PROGRAM MAIN
VAR_OUTPUT //globally readable, but only modifiable by MAIN
	outputBuffer : ARRAY[Surface.LEFT..Surface.RIGHT] OF Bundle;
	outputBufferPass, outputBufferFail : Bundle;
	numOutputBundles : USINT := 0;
	
	bundleIn : Bundle;
	bundleOut : Bundle;
	
	start : BOOL;
	
	ready : BOOL;
	busy : BOOL;
	done : BOOL;
	error : BOOL;
	backlog : BOOL;
	
	stop : BOOL;
	execute : BOOL;
	hold : BOOL;
	reset : BOOL;
	
	localTime : TIMESTRUCT;
	
	pmlModeString : STRING;
	pmlStateString : STRING;
END_VAR
VAR
	clearPassBuffer, clearFailBuffer AT %I* : BOOL;
	receiverStruct : AdsData;
	
	//ETA is not strictly required, area will process bundle even if it is not in ETA arrays
	expectedBundles : ARRAY[0..GVL.maxQueue] OF STRING; //bundles expected to arrive
	expectedArrivals : ARRAY[0..GVL.maxQueue] OF TIMESTRUCT; //bundles expected to arrive
	numEtaBundles : INT;
	
	//parallel arrays - bundle, bypass
	numBundles : INT;
	bundlesQueue : ARRAY[0..GVL.maxQueue] OF Bundle;
	bundlesBypass : ARRAY[0..GVL.maxQueue] OF BOOL;
END_VAR
VAR
	//spacerRecollector : PackagerFreeAsync;
	//paperSection : PaperEx;
	//cardboardCornerGuardSection : CardboardCornerGuardEx;
	//chipboardSection : ChipboardEx;
	woodBunkSection : WoodBunkEx;
	//outputSection : AreaOutputEx;	
END_VAR
VAR
	fbLocalSystemTime : FB_LocalSystemTime;
	dbLogger : SqlDatabaseAccessor;
	conveyorController : ConveyorControlUnit;
	
	pmlState : E_PMLState;
	pmlCommand : E_PMLCommand;
	pmlStateMachine : PML_StateMachine;
	
	pmlModeRequest : E_PMLCustomUnitMode := ePMLCustomUnitMode_Production;
	pmlMode : E_PMLCustomUnitMode;
	pmlModeManager : PML_UnitModeManager;
END_VAR
VAR //these variables are only tracked for HMI
	sectionsBusy : ARRAY[0..SectionEnum.size] OF BOOL;
	sectionsIterator : ARRAY[0..SectionEnum.size] OF INT;
END_VAR

(*
ready := paperSection.ready; //if A2 is not ready, dispatch controller must block operator from sending bundles here
busy := paperSection.busy OR cardboardCornerGuardSection.busy OR chipboardSection.busy OR woodBunkSection.busy OR outputSection.busy;
done := outputSection.done;
backlog := numBundlesQueue > 5;
*)

CallHardware(); //start program with CallHardware()
SetupHardware(); //set bEnables, setup material holder slots, etc

initialize();

fillBundlesQueue();

SizeCheck();
getLocalTime();

AdsClient( //PLC-PLC comms
	ServerNetId:= , 
	ServerPort:= , 
	bBusy=> , 
	err=> , 
	errid=> , 
	localPrgName=> , 
	localNetId=> , 
	localPort=> , 
	socketReady=> , 
	remoteAccessPrefix=> );
	
TcpServer1Vision( //PLC-Vision comms
	ServerNetId:= , 
	ServerAdr:= , 
	ServerPort:= , 
	busy=> , 
	error=> , 
	errorId=> , 
	bytesReceived=> , 
	connected=> , 
	receiveStruct=> );
	
runPML();

IF AdsClient.fetchData(receiverStruct) THEN
	interpretTransmission(receiverStruct);
END_IF


IF ready AND BundleIsValid(bundleIn) THEN
	receive();
END_IF


IF clearPassBuffer OR clearFailBuffer THEN
	transfer();
	shiftBundles();
END_IF

dbLogger();

conveyorController(conveyors := conveyorsArr);
CallHardware(); //start program with CallHardware()

METHOD fillBundlesQueue : BOOL
VAR
	i : INT;
END_VAR
IF NOT start THEN //for HMI testing only, remove for production
	FOR i:=0 TO GVL.maxQueue BY 1 DO
		bundlesQueue[i].id := TO_STRING(i);
	END_FOR
	
	start := TRUE;
END_IF
END_METHOD

METHOD PRIVATE getLocalTime : BOOL
fbLocalSystemTime(
	sNetID:= '', 
	bEnable:= TRUE, 
	dwCycle:= , 
	dwOpt:= , 
	tTimeout:= , 
	bValid=> , 
	systemTime=> localTime, 
	tzID=> );
	
getLocalTime := TRUE;
END_METHOD

METHOD PRIVATE initialize : BOOL
//paperSection.connectTo(ADR(cardboardCornerGuardSection));
//cardboardCornerGuardSection.connectTo(ADR(chipboardSection));
//chipboardSection.connectTo(ADR(woodBunkSection));
woodBunkSection.connectTo(0); //(ADR(outputSection));
//connecting to 0 means no next section

//paperSection.sectionID := SectionEnum.PAPER;
//cardboardCornerGuardSection.sectionID := SectionEnum.CARDBOARD_CORNERGUARD;
//chipboardSection.sectionID := SectionEnum.CHIPBOARD;
woodBunkSection.sectionID := SectionEnum.WOOD_BUNK;
//outputSection.sectionID := SectionEnum.OUTPUT;

(*
	paperSection.pNextSection := ADR(cardboardCornerGuardSection);
	cardboardCornerGuardSection.accessNextSection := ADR(chipboardSection);
	chipboardSection.accessNextSection := ADR(woodBunkSection);
	woodBunkSection.accessNextSection := ADR(outputSection);
	outputSection.accessNextSection := 0;
*)

initialize := TRUE;
END_METHOD

METHOD PRIVATE interpretTransmission : BOOL
VAR_INPUT
	data : REFERENCE TO AdsData;
END_VAR
VAR
	i : INT;
END_VAR
CASE data.description OF
	EventsEnum.BUNDLE_IN:
		MEMCPY(ADR(bundleIn), ADR(data.binaryData), SIZEOF(bundleIn));
			
	EventsEnum.BUNDLE_ETA:
		MEMCPY(ADR(expectedBundles[numEtaBundles]), ADR(data.binaryData), SIZEOF(expectedBundles[numEtaBundles]));
		expectedArrivals[numEtaBundles] := data.timestamp;
		
END_CASE
END_METHOD

METHOD maintenance : BOOL
VAR_INPUT
END_VAR
END_METHOD

METHOD PRIVATE process : BOOL
(*
full parallel processsing
all sections may operate concurrently on any bundle
*)
(*
paperSection(
	enable:= run[SectionEnum.PAPER], 
	bundlesQueue:= bundlesQueue, 
	bundlesBypass:= bundlesBypass,
	bundleOut=> , 
	bypass=> , 
	ready=> , 
	busy=> sectionsBusy[SectionEnum.PAPER], 
	done=> , 
	error=> , 
	backlog=> ,
	iBundle=> sectionsIterator[SectionEnum.PAPER],
	iPair=> );
	
cardboardCornerGuardSection(
	enable:= run[SectionEnum.CARDBOARD_CORNERGUARD],
	bundlesQueue:= bundlesQueue, 
	bundlesBypass:= bundlesBypass,
	bundleOut=> ,
	bypass=> , 
	ready=> , 
	busy=> sectionsBusy[SectionEnum.CARDBOARD_CORNERGUARD], 
	done=> , 
	error=> , 
	backlog=> ,
	iBundle=> sectionsIterator[SectionEnum.CARDBOARD_CORNERGUARD],
	iPair=> );

chipboardSection(
	enable:= run[SectionEnum.CHIPBOARD],
	bundlesQueue:= bundlesQueue, 
	bundlesBypass:= bundlesBypass, 
	bundleOut=> ,
	bypass=> , 
	ready=> , 
	busy=> sectionsBusy[SectionEnum.CHIPBOARD], 
	done=> , 
	error=> , 
	backlog=> ,
	iBundle=> sectionsIterator[SectionEnum.CHIPBOARD],
	iPair=> );
*)

(*
woodBunkSection(
	enable:= run[SectionEnum.WOOD_BUNK],
	bundlesQueue:= bundlesQueue, 
	bundlesBypass:= bundlesBypass, 
	bundleOut=> ,
	bypass=> , 
	ready=> , 
	busy=> sectionsBusy[SectionEnum.WOOD_BUNK], 
	done=> , 
	error=> , 
	backlog=> ,
	iBundle=> sectionsIterator[SectionEnum.WOOD_BUNK],
	iPair=> );
*)
(*
outputSection(
	enable:= run[SectionEnum.OUTPUT],
	bundlesQueue:= bundlesQueue, 
	bundlesBypass:= bundlesBypass,
	outputBuffer:= outputBuffer,
	bundleOut=> , 
	bypass=> , 
	ready=> , 
	busy=> sectionsBusy[SectionEnum.OUTPUT],
	done=> , 
	error=> , 
	backlog=> ,
	iBundle=> sectionsIterator[SectionEnum.OUTPUT],
	iPair=> );
*)
END_METHOD

METHOD PRIVATE processLLD : BOOL
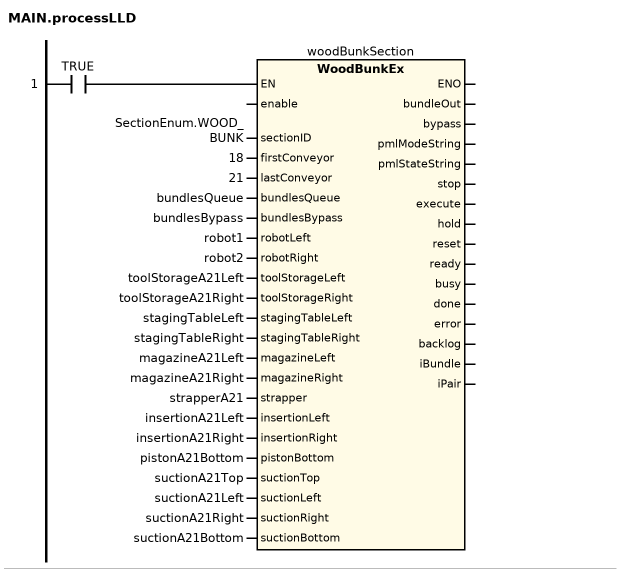
// NETWORK 1
woodBunkSection(
    sectionID := SectionEnum.WOOD_BUNK,
    firstConveyor := 18,
    lastConveyor := 21,
    bundlesQueue := bundlesQueue,
    bundlesBypass := bundlesBypass,
    robotLeft := robot1,
    robotRight := robot2,
    toolStorageLeft := toolStorageA21Left,
    toolStorageRight := toolStorageA21Right,
    stagingTableLeft := stagingTableLeft,
    stagingTableRight := stagingTableRight,
    magazineLeft := magazineA21Left,
    magazineRight := magazineA21Right,
    strapper := strapperA21,
    insertionLeft := insertionA21Left,
    insertionRight := insertionA21Right,
    pistonBottom := pistonA21Bottom,
    suctionTop := suctionA21Top,
    suctionLeft := suctionA21Left,
    suctionRight := suctionA21Right,
    suctionBottom := suctionA21Bottom); // WoodBunkEx
END_METHOD

METHOD PRIVATE ps_AbortCondition : BOOL
VAR_INPUT
END_VAR
END_METHOD

METHOD PRIVATE ps_Aborted : BOOL
VAR_INPUT
END_VAR
END_METHOD

METHOD PRIVATE ps_Aborting : BOOL
VAR_INPUT
END_VAR
END_METHOD

METHOD PRIVATE ps_Clearing : BOOL
VAR_INPUT
END_VAR
END_METHOD

METHOD PRIVATE ps_Complete : BOOL
VAR_INPUT
END_VAR
END_METHOD

METHOD PRIVATE ps_Completing : BOOL
VAR_INPUT
END_VAR
END_METHOD

METHOD PRIVATE ps_Execute : BOOL
VAR_INPUT
END_VAR
VAR_OUTPUT
	error : BOOL;
END_VAR
CASE pmlMode OF
	0: //invalid mode
	ePMLCustomUnitMode_Production:		ps_Execute := process();
	ePMLCustomUnitMode_Maintenance:		maintenance();
	ePMLCustomUnitMode_Manual:			//
	ePMLCustomUnitMode_SemiAuto:		ps_Execute := process(); //manually step bundle into area - sections may be auto while area is semi-auto
END_CASE
END_METHOD

METHOD PRIVATE ps_Held : BOOL
VAR_INPUT
END_VAR
END_METHOD

METHOD PRIVATE ps_HoldCondition : BOOL
VAR_INPUT
END_VAR
END_METHOD

METHOD PRIVATE ps_Holding : BOOL
VAR_INPUT
END_VAR
END_METHOD

METHOD PRIVATE ps_Idle : BOOL
VAR_INPUT
END_VAR
(*
IF BundleIsValid(currentBundle) THEN
	ps_Idle := TRUE;
	done := FALSE;
END_IF
*)

ps_Idle := TRUE; (*start section input*)
END_METHOD

METHOD PRIVATE ps_Resetting : BOOL
VAR_INPUT
END_VAR
END_METHOD

METHOD PRIVATE ps_Starting : BOOL
VAR_INPUT
END_VAR
END_METHOD

METHOD PRIVATE ps_StopCondition : BOOL
VAR_INPUT
END_VAR
END_METHOD

METHOD PRIVATE ps_Stopped : BOOL
VAR_INPUT
END_VAR
END_METHOD

METHOD PRIVATE ps_Stopping : BOOL
VAR_INPUT
END_VAR
END_METHOD

METHOD PRIVATE ps_SuspendCondition : BOOL
VAR_INPUT
END_VAR
END_METHOD

METHOD PRIVATE ps_Suspended : BOOL
VAR_INPUT
END_VAR
END_METHOD

METHOD PRIVATE ps_Suspending : BOOL
VAR_INPUT
END_VAR
END_METHOD

METHOD PRIVATE ps_Unholding : BOOL
VAR_INPUT
END_VAR
END_METHOD

METHOD PRIVATE ps_Unsuspending : BOOL
VAR_INPUT
END_VAR
END_METHOD

{attribute 'TcRpcEnable'}
METHOD PRIVATE receive : BOOL
VAR
	i : INT;
	shiftIndex : INT := -1;
	invalidBundle : Bundle;
END_VAR
FOR i:=0 TO GVL.maxQueue BY 1 DO //find the bundle in the ETA queue
	IF expectedBundles[i] = bundleIn.id THEN
		shiftIndex := i;
		EXIT;
	END_IF
END_FOR

IF shiftIndex > -1 THEN //if the bundle is found in the ETA queue, shift everything down
	MEMMOVE(
		ADR(expectedBundles[shiftIndex]), 
		ADR(expectedBundles[shiftIndex + 1]), 
		SIZEOF(STRING) * TO_UINT(GVL.maxQueue - shiftIndex));
		
	MEMMOVE(
		ADR(expectedArrivals[shiftIndex]), 
		ADR(expectedArrivals[shiftIndex + 1]), 
		SIZEOF(TIMESTRUCT) * TO_UINT(GVL.maxQueue - shiftIndex) );
		
	numEtaBundles := numEtaBundles - 1;
END_IF

FOR i:=0 TO GVL.maxQueue BY 1 DO
	IF BundleIsValid(bundlesQueue[i]) AND NOT bundlesBypass[i] THEN
		bundlesQueue[i] := bundleIn;
		bundlesBypass[i] := FALSE;
		
		receive := TRUE;
		RETURN;
	END_IF
END_FOR

IF NOT receive THEN
	error := TRUE;
END_IF
END_METHOD

METHOD PRIVATE runPML : BOOL
(*
PackML
	state machine for packaging applications - see Tc3_PackML_V2 library on InfoSys
	
	final states - wait for an input or condition and command to new state
	intermediate states - complete a task and call pmlStateMachine.M_StateComplete() to advance to next state
	
the following states currently use the same logic (albeit in different methods), implementation may change later
	ps_Stopping() and ps_Aborting()
	ps_Resetting() and ps_Clearing()
	
STOP - controlled stop **with intent to shutdown or vacate for extended time** induced by operator/HMI - otherwise use HOLD
ABORT - emergency stop due to machine errors


HOLD - minor local issues
SUSPEND - external issues

EXECUTE - major control logic
	different modes may require different tasks
	create methods as required for different modes, then call the correct method in ps_Completing()
	can be commanded to STOP, ABORT, HOLD, or SUSPEND at any point
COMPLETING - process complete, move product out of system and finish transition to COMPLETED

the implementation below can be copied to all POUs that use a PackML state machine
the individual ps_< > methods need to be implemented for the specific application
*)
IF ps_AbortCondition() THEN //abort condition
	pmlCommand := ePMLCommand_Abort;
ELSIF ps_StopCondition() THEN //stop condition
	pmlCommand := ePMLCommand_Stop;
END_IF

CASE pmlState OF
	0 (*ePMLState_Undefined*): //default state on startup
		pmlCommand := ePMLCommand_Stop;
		
	ePMLState_Stopping:
		IF ps_Stopping() THEN
			pmlStateMachine.M_StateComplete();
		END_IF
		
	ePMLState_Stopped:
		IF ps_Stopped() THEN
			pmlCommand := ePMLCommand_Reset;
		END_IF
	
    ePMLState_Resetting:
		IF ps_Resetting() THEN
			pmlStateMachine.M_StateComplete();
		END_IF
		
	ePMLState_Idle:
		IF ps_Idle() THEN
			pmlCommand := ePMLCommand_Start;
		END_IF		
	
	ePMLState_Starting:
		IF ps_Starting() THEN
			pmlStateMachine.M_StateComplete();
		END_IF
	
	ePMLState_Execute: //check the conditions in order of their priority, currently HOLD has the highest priority
		IF ps_HoldCondition() THEN
			pmlCommand := ePMLCommand_Hold;
			
		ELSIF ps_SuspendCondition() THEN
			pmlCommand := ePMLCommand_Suspend;			
		
		ELSIF ps_Execute(error => error) THEN //ps_Execute.error => THIS^.error
			pmlStateMachine.M_StateComplete();
			pmlCommand := ePMLCommand_Complete;
		END_IF
		
	ePMLState_Completing:
		IF ps_Completing() THEN
			pmlStateMachine.M_StateComplete();
		END_IF
	
	ePMLState_Complete:
		IF ps_Complete() THEN
			pmlCommand := ePMLCommand_Reset;
		END_IF
	
	ePMLState_Holding:
		IF ps_Holding() THEN
			pmlStateMachine.M_StateComplete();
		END_IF
	
	ePMLState_Held:
		IF NOT hold THEN
			pmlCommand := ePMLCommand_Unhold;
		END_IF
	
	ePMLState_Unholding:
		IF ps_Unholding() THEN
			pmlStateMachine.M_StateComplete(); //release all pause commands and IO
		END_IF
		
	ePMLState_Suspending: //based on next section conditions
		IF ps_Suspending() THEN
			pmlStateMachine.M_StateComplete();
		END_IF
		
	ePMLState_Suspended: //based on next section conditions
		IF ps_Suspended() THEN
			pmlCommand := ePMLCommand_Unsuspend;
		END_IF
	
	ePMLState_Unsuspending: //based on next section conditions
		IF ps_Unsuspending() THEN
			pmlStateMachine.M_StateComplete();
		END_IF
	
	ePMLState_Aborting:
		IF ps_Aborting() THEN
			pmlStateMachine.M_StateComplete();
		END_IF
	
	ePMLState_Aborted:
		IF ps_Aborted() THEN
			pmlCommand := ePMLCommand_Clear;
		END_IF
	
	ePMLState_Clearing:
		IF ps_Clearing() THEN
			pmlStateMachine.M_StateComplete();
		END_IF
	
END_CASE
END_METHOD

METHOD shiftBundles : BOOL
VAR_INPUT
END_VAR
//shift down parallel arrays
MEMMOVE(ADR(bundlesQueue[0]), ADR(bundlesQueue[1]), SIZEOF(Bundle) * TO_UINT(GVL.maxQueue));
MEMMOVE(ADR(bundlesBypass[0]), ADR(bundlesBypass[1]), SIZEOF(BOOL) * TO_UINT(GVL.maxQueue));

//decrement each section's iterator to realign with their correct bundle
//paperSection.shiftIterator();
//cardboardCornerGuardSection.shiftIterator();
//chipboardSection.shiftIterator();
woodBunkSection.shiftIterator();
//outputSection.shiftIterator();
END_METHOD

METHOD PRIVATE transfer : BOOL
VAR
	i : INT;
END_VAR
//send TCP/ADS transmission back to Dispatch once bundle is removed from the plant

IF clearPassBuffer THEN
	dbLogger.queueEvent(event:= EventsEnum.BUNDLE_OUT); //modify to include bundle ID
	//outputBufferPass := GVL.nullBundle;
	MEMSET(ADR(outputBufferPass), 0, SIZEOF(outputBufferPass));
END_IF

IF clearFailBuffer THEN
	dbLogger.queueEvent(event:= EventsEnum.BUNDLE_OUT); //modify to include bundle ID
	//outputBufferFail := GVL.nullBundle;
	MEMSET(ADR(outputBufferFail), 0, SIZEOF(outputBufferFail));
END_IF
END_METHOD

END_PROGRAM

(* stored: Version 1.1.0.1, ProductVersion 3.1.4024.11
   POU MAIN: Id {f8ea2e52-8cdd-4c5a-a5f9-4c8d8a3c6a2c}, SpecialFunc None
   Folder PML Conditions: Id {c04cfa90-34d0-4dce-a54d-25d4cc1b429e}
   Folder PML States: Id {6ef5f588-dba8-43b6-aecd-30cae96b064d}
   Folder Process Modes: Id {8d1d624d-f207-4b80-ae71-4f41b10197eb}
   Folder Setup: Id {766689c6-4b05-4d8b-a8a4-3bf5c2750aa3}
   Method fillBundlesQueue: Id {73fc04c3-3b20-4b90-b668-e45a325d9c2c}
   Method getLocalTime: Id {b9dfd14b-062f-4ab4-b051-cd1816451bba}
   Method initialize: Id {1af4c629-041d-43ca-9e16-2266f17c58c8}
   Method interpretTransmission: Id {04aa253b-ab0d-41b0-b6b2-443fd8efedd5}
   Method maintenance: Id {0fc159f6-b7a4-4008-822a-e6f2dd60b8f1}
   Method process: Id {f9da02b9-c065-4582-840f-d291dad1e576}
   Method processLLD: Id {042e9a05-7085-4896-a772-b3d42ff1357c}
   Method ps_AbortCondition: Id {2bb22b37-bb31-4cf8-9360-ad8974e4345a}
   Method ps_Aborted: Id {8b7e8913-d6a1-4d11-8ef4-5de3678c0038}
   Method ps_Aborting: Id {2cfb75cc-c590-4cea-9c9e-baef234b3390}
   Method ps_Clearing: Id {2e0869f6-c4a9-4781-8ad2-74da1ae357b5}
   Method ps_Complete: Id {b669e02a-682b-4740-906b-0def158a3c63}
   Method ps_Completing: Id {d62eb91d-4af1-4f38-ab45-c3b8a61c00fe}
   Method ps_Execute: Id {1599d25a-dab9-4ec4-92fd-68ba4e793876}
   Method ps_Held: Id {95c54fec-4967-44f4-be8f-1e853d267e68}
   Method ps_HoldCondition: Id {ede1d647-a96e-40da-9b59-0807c117e213}
   Method ps_Holding: Id {c19fae67-2974-4ceb-8f46-951138e6d029}
   Method ps_Idle: Id {d98cd4ab-14fc-4d54-b00b-761967e4ce59}
   Method ps_Resetting: Id {800fa30c-d995-43ee-a200-3b63842e0a79}
   Method ps_Starting: Id {63620e6e-9309-4b45-8ae4-a18a69032f6f}
   Method ps_StopCondition: Id {3958b83a-de5c-49c7-92a1-84b37d19df0a}
   Method ps_Stopped: Id {842f7be6-f686-4ed8-9cf9-1ceced765cfd}
   Method ps_Stopping: Id {e0fa46b1-b44a-4e23-a32e-d1b02ace1ef6}
   Method ps_SuspendCondition: Id {ac03eab2-8477-4493-9499-38a84b2dca7e}
   Method ps_Suspended: Id {977bb7ef-1ea7-4419-8df9-c453c72a4fd4}
   Method ps_Suspending: Id {5beb683b-6fd3-4fc2-9a12-97f55383c8c4}
   Method ps_Unholding: Id {290593bb-af9d-4c36-8150-3909fafedce7}
   Method ps_Unsuspending: Id {cb22f287-33db-44c9-9aac-845a4a32160a}
   Method receive: Id {2de20b6b-9727-4ca1-a75e-22c752a3c085}
   Method runPML: Id {70af2742-8e75-45b6-8123-d51f2e8f6038}
   Method shiftBundles: Id {5473c570-b523-4be9-bf64-c8f58c1af44e}
   Method transfer: Id {a55e1076-0c29-4969-952a-05c194ea9e2d} *)
